TYPE E_DispenserState :
(
	Idle,
	Preparing,
	Dispensing
)USINT;
END_TYPE

(* stored: Version 1.1.0.1, ProductVersion 3.1.4024.5
   DUT E_DispenserState: Id {d8733d62-f198-48ef-a2d7-c9e6561e5529} *)
